{attribute 'GeneratedUsingTerminal: EL2642-0000-0016'}
{attribute addProperty BoxType "EL2642-0000-0016"}
{attribute addProperty Id "Device_statusAT %I*Device_status_8568DBCA3"}
{attribute addProperty CRC "1250970053"}
{attribute addProperty Size "3"}
TYPE DO_Inputs_Device_4A9049C5 EXTENDS InputBase_8311D824 :
STRUCT
	{attribute addProperty Name "Device_status"}
	Device_status AT %I* : Device_status_8568DBCA;
END_STRUCT
END_TYPE

(* stored: Version 1.2.0.0, ProductVersion 3.1.4024.9
   DUT DO_Inputs_Device_4A9049C5: Id {497f4450-89e9-4e98-a819-97de35293014} *)
